TYPE ST_System_LA_Stellwert :
STRUCT

END_STRUCT
END_TYPE

(* stored: Version 1.1.0.1, ProductVersion 3.1.4024.9
   DUT ST_System_LA_Stellwert: Id {a3b3c2a9-16ef-4e96-95b5-8059597229b2} *)
